(*
  string concat for length > 255
*)
FUNCTION f_Builder : Bool
VAR_INPUT
  pInString   : POINTER TO STRING;
  pOutString  : POINTER TO STRING(32767);
  //pOutString  : POINTER TO STRING(16384);
  fLength     : INT;
END_VAR
VAR
  Counter     : DINT;
  pInWork     : POINTER TO BYTE;
  pOutWork    : POINTER TO BYTE;
END_VAR

pOutWork := pOutString;
pInWork := pInString;
Counter := 0;

(*check termination*)
WHILE (pOutWork^ <> 0) AND
      (Counter < 32767)
DO
  Counter := Counter + 1;
  pOutWork := pOutWork + 1;
END_WHILE

(* append only if data fits into output *)
IF (Counter + fLength < 32767)
THEN

  (* append data *)
  FOR Counter := 1 TO fLength
  DO
    pOutWork^ := pInWork^;
    pOutWork := pOutWork + 1;
    pInWork := pInWork + 1;
  END_FOR

  (* terminate *)
  pOutWork := pOutWork + 1;
  pOutWork^ := 0;
END_IF

END_FUNCTION

(* stored: Version 1.1.0.1, ProductVersion 3.1.4022.18
   POU f_Builder: Id {77abc0a8-921c-4470-93e3-900bef91b873}, SpecialFunc None *)
